(*

## Short summary
This class provides assert statements for bytes.

.. <legal notes>

legal notes
=================
| SPDX-FileCopyrightText: © 2022 ekvip automation GmbH <info@ekvip.de>
| SPDX-License-Identifier: Apache-2.0
| For details check: Apache-2.0_

.. _Apache-2.0: https://www.apache.org/licenses/LICENSE-2.0

.. </legal notes>



*)

{attribute 'reflection'}
FUNCTION_BLOCK INTERNAL ByteAssertions EXTENDS AbstractAssertion IMPLEMENTS IByteAssertions
VAR
END_VAR
VAR CONSTANT
	(* least significant bit *)
	LSB	:BYTE := 16#01;
	(* most significant bit *)
	MSB :BYTE := 16#80;
END_VAR

(*

## Short summary
This assertion method checks if the result current value bitwise ``AND`` mask is equal to the expected value

.. <legal notes>

legal notes
=================
| SPDX-FileCopyrightText: © 2022 ekvip automation GmbH <info@ekvip.de>
| SPDX-License-Identifier: Apache-2.0
| For details check: Apache-2.0_

.. _Apache-2.0: https://www.apache.org/licenses/LICENSE-2.0

.. </legal notes>



*)

METHOD andMaskIsEqualTo
VAR_INPUT
	(* current value to check *)
	currentValue	:BYTE;
	(* 2nd operand for bitwise operation *)
	mask			:BYTE;
	(* expected result after masking *)
	expectedValue	:BYTE;
	(* message if the assertion is false *)
	message			:AssertMessage;
END_VAR
IF ((currentValue AND mask) <> expectedValue) THEN
	THIS^.assertionWasWrong(message, THIS^.getDebugInfo('andMaskIsEqualTo'));
END_IF
END_METHOD

(*

## Short summary
This assertion method checks if the result current value bitwise ``AND`` mask
is not equal to the unexpected value

.. <legal notes>

legal notes
=================
| SPDX-FileCopyrightText: © 2022 ekvip automation GmbH <info@ekvip.de>
| SPDX-License-Identifier: Apache-2.0
| For details check: Apache-2.0_

.. _Apache-2.0: https://www.apache.org/licenses/LICENSE-2.0

.. </legal notes>



*)

METHOD andMaskIsNotEqualTo
VAR_INPUT
	(* current value to check *)
	currentValue	:BYTE;
	(* 2nd operand for bitwise operation *)
	mask			:BYTE;
	(* unexpected result after masking *)
	unexpectedValue	:BYTE;
	(* message if the assertion is false *)
	message			:AssertMessage;
END_VAR
IF ((currentValue AND mask) = unexpectedValue) THEN
	THIS^.assertionWasWrong(message, THIS^.getDebugInfo('andMaskIsNotEqualTo'));
END_IF
END_METHOD

(*

## Short summary
This assertion method checks if the selected bit of current value
is equal to the expected value

.. <legal notes>

legal notes
=================
| SPDX-FileCopyrightText: © 2022 ekvip automation GmbH <info@ekvip.de>
| SPDX-License-Identifier: Apache-2.0
| For details check: Apache-2.0_

.. _Apache-2.0: https://www.apache.org/licenses/LICENSE-2.0

.. </legal notes>



*)

METHOD bitXIsEqualTo
VAR_INPUT
	(* current value to check *)
	currentValue	:BYTE;
	(* number of bit to check *)
	number			:BitNumberByte;
	(* expected value of bit *)
	expectedValue	:BOOL;
	(* message if the assertion is false *)
	message			:AssertMessage;
END_VAR
IF (
	TO_BOOL(
		TO_BYTE(SHL(THIS^.LSB, number))
		AND currentValue
	) <> expectedValue
) THEN
	THIS^.assertionWasWrong(message, THIS^.getDebugInfo('bitXIsEqualTo'));
END_IF
END_METHOD

(*

## Short summary
This assertion method checks if the selected bit of current value
is not equal to the unexpected value

.. <legal notes>

legal notes
=================
| SPDX-FileCopyrightText: © 2022 ekvip automation GmbH <info@ekvip.de>
| SPDX-License-Identifier: Apache-2.0
| For details check: Apache-2.0_

.. _Apache-2.0: https://www.apache.org/licenses/LICENSE-2.0

.. </legal notes>



*)

METHOD bitXIsNotEqualTo
VAR_INPUT
	(* current value to check *)
	currentValue	:BYTE;
	(* number of bit to check *)
	number			:BitNumberByte;
	(* unexpected value of bit *)
	unexpectedValue	:BOOL;
	(* message if the assertion is false *)
	message			:AssertMessage;
END_VAR
IF (
	TO_BOOL(
		TO_BYTE(SHL(THIS^.LSB, number))
		AND currentValue
	) = unexpectedValue
) THEN
	THIS^.assertionWasWrong(message, THIS^.getDebugInfo('bitXIsNotEqualTo'));
END_IF
END_METHOD

(*

## Short summary
This assertion method checks if the selected bit of current value
is set

.. <legal notes>

legal notes
=================
| SPDX-FileCopyrightText: © 2022 ekvip automation GmbH <info@ekvip.de>
| SPDX-License-Identifier: Apache-2.0
| For details check: Apache-2.0_

.. _Apache-2.0: https://www.apache.org/licenses/LICENSE-2.0

.. </legal notes>



*)

METHOD bitXIsSet
VAR_INPUT
	(* current value to check *)
	currentValue	:BYTE;
	(* number of bit to check *)
	number			:BitNumberByte;
	(* message if the assertion is false *)
	message			:AssertMessage;
END_VAR
IF (
	NOT TO_BOOL(
		TO_BYTE(SHL(THIS^.LSB, number))
		AND currentValue
	)
) THEN
	THIS^.assertionWasWrong(message, THIS^.getDebugInfo('bitXIsSet'));
END_IF
END_METHOD

(*

## Short summary
This assertion method checks if the selected bit of current value
is unset

.. <legal notes>

legal notes
=================
| SPDX-FileCopyrightText: © 2022 ekvip automation GmbH <info@ekvip.de>
| SPDX-License-Identifier: Apache-2.0
| For details check: Apache-2.0_

.. _Apache-2.0: https://www.apache.org/licenses/LICENSE-2.0

.. </legal notes>



*)

METHOD bitXIsUnset
VAR_INPUT
	(* current value to check *)
	currentValue	:BYTE;
	(* number of bit to check *)
	number			:BitNumberByte;
	(* message if the assertion is false *)
	message			:AssertMessage;
END_VAR
IF (
	TO_BOOL(
		TO_BYTE(SHL(THIS^.LSB, number))
		AND currentValue
	)
) THEN
	THIS^.assertionWasWrong(message, THIS^.getDebugInfo('bitXIsUnset'));
END_IF
END_METHOD

(*

## Short summary
This abstract property returns the class name of the concrete object, 
It's for debugging purpose

.. <legal notes>

legal notes
=================
| SPDX-FileCopyrightText: © 2022 ekvip automation GmbH <info@ekvip.de>
| SPDX-License-Identifier: Apache-2.0
| For details check: Apache-2.0_

.. _Apache-2.0: https://www.apache.org/licenses/LICENSE-2.0

.. </legal notes>

*)

PROPERTY className :CNM_AbstractObject.ClassName
GET
className := 'CNM_Assertor.ByteAssertions';
END_GET
END_PROPERTY

(*

## Short summary
This assertion method checks if the least significant bit of current value
is equal to the expected value

.. <legal notes>

legal notes
=================
| SPDX-FileCopyrightText: © 2022 ekvip automation GmbH <info@ekvip.de>
| SPDX-License-Identifier: Apache-2.0
| For details check: Apache-2.0_

.. _Apache-2.0: https://www.apache.org/licenses/LICENSE-2.0

.. </legal notes>



*)

METHOD lsbIsEqualTo
VAR_INPUT
	(* current value to check *)
	currentValue	:BYTE;
	(* expected value of lsb *)
	expectedValue	:BOOL;
	(* message if the assertion is false *)
	message			:AssertMessage;
END_VAR
IF (TO_BOOL(currentValue AND THIS^.LSB) <> expectedValue) THEN
	THIS^.assertionWasWrong(message, THIS^.getDebugInfo('lsbIsEqualTo'));
END_IF
END_METHOD

(*

## Short summary
This assertion method checks if the least significant bit of current value
is not equal to the unexpected value

.. <legal notes>

legal notes
=================
| SPDX-FileCopyrightText: © 2022 ekvip automation GmbH <info@ekvip.de>
| SPDX-License-Identifier: Apache-2.0
| For details check: Apache-2.0_

.. _Apache-2.0: https://www.apache.org/licenses/LICENSE-2.0

.. </legal notes>



*)

METHOD lsbIsNotEqualTo
VAR_INPUT
	(* current value to check *)
	currentValue	:BYTE;
	(* unexpected value of lsb *)
	unexpectedValue	:BOOL;
	(* message if the assertion is false *)
	message			:AssertMessage;
END_VAR
IF (TO_BOOL(currentValue AND THIS^.LSB) = unexpectedValue) THEN
	THIS^.assertionWasWrong(message, THIS^.getDebugInfo('lsbIsNotEqualTo'));
END_IF
END_METHOD

(*

## Short summary
This assertion method checks if the least significant bit of current value
is set

.. <legal notes>

legal notes
=================
| SPDX-FileCopyrightText: © 2022 ekvip automation GmbH <info@ekvip.de>
| SPDX-License-Identifier: Apache-2.0
| For details check: Apache-2.0_

.. _Apache-2.0: https://www.apache.org/licenses/LICENSE-2.0

.. </legal notes>



*)

METHOD lsbIsSet
VAR_INPUT
	(* current value to check *)
	currentValue	:BYTE;
	(* message if the assertion is false *)
	message			:AssertMessage;
END_VAR
IF (NOT TO_BOOL(currentValue AND THIS^.LSB)) THEN
	THIS^.assertionWasWrong(message, THIS^.getDebugInfo('lsbIsSet'));
END_IF
END_METHOD

(*

## Short summary
This assertion method checks if the least significant bit of current value
is unset

.. <legal notes>

legal notes
=================
| SPDX-FileCopyrightText: © 2022 ekvip automation GmbH <info@ekvip.de>
| SPDX-License-Identifier: Apache-2.0
| For details check: Apache-2.0_

.. _Apache-2.0: https://www.apache.org/licenses/LICENSE-2.0

.. </legal notes>



*)

METHOD lsbIsUnset
VAR_INPUT
	(* current value to check *)
	currentValue	:BYTE;
	(* message if the assertion is false *)
	message			:AssertMessage;
END_VAR
IF (TO_BOOL(currentValue AND THIS^.LSB)) THEN
	THIS^.assertionWasWrong(message, THIS^.getDebugInfo('lsbIsUnset'));
END_IF
END_METHOD

(*

## Short summary
This assertion method checks if the most significant bit of current value
is equal to the expected value

.. <legal notes>

legal notes
=================
| SPDX-FileCopyrightText: © 2022 ekvip automation GmbH <info@ekvip.de>
| SPDX-License-Identifier: Apache-2.0
| For details check: Apache-2.0_

.. _Apache-2.0: https://www.apache.org/licenses/LICENSE-2.0

.. </legal notes>



*)

METHOD msbIsEqualTo
VAR_INPUT
	(* current value to check *)
	currentValue	:BYTE;
	(* expected value of msb *)
	expectedValue	:BOOL;
	(* message if the assertion is false *)
	message			:AssertMessage;
END_VAR
IF (TO_BOOL(currentValue AND THIS^.MSB) <> expectedValue) THEN
	THIS^.assertionWasWrong(message, THIS^.getDebugInfo('msbIsEqualTo'));
END_IF
END_METHOD

(*

## Short summary
This assertion method checks if the most significant bit of current value
is not equal to the unexpected value

.. <legal notes>

legal notes
=================
| SPDX-FileCopyrightText: © 2022 ekvip automation GmbH <info@ekvip.de>
| SPDX-License-Identifier: Apache-2.0
| For details check: Apache-2.0_

.. _Apache-2.0: https://www.apache.org/licenses/LICENSE-2.0

.. </legal notes>



*)

METHOD msbIsNotEqualTo
VAR_INPUT
	(* current value to check *)
	currentValue	:BYTE;
	(* unexpected value of msb *)
	unexpectedValue	:BOOL;
	(* message if the assertion is false *)
	message			:AssertMessage;
END_VAR
IF (TO_BOOL(currentValue AND THIS^.MSB) = unexpectedValue) THEN
	THIS^.assertionWasWrong(message, THIS^.getDebugInfo('msbIsNotEqualTo'));
END_IF
END_METHOD

(*

## Short summary
This assertion method checks if the most significant bit of current value
is set

.. <legal notes>

legal notes
=================
| SPDX-FileCopyrightText: © 2022 ekvip automation GmbH <info@ekvip.de>
| SPDX-License-Identifier: Apache-2.0
| For details check: Apache-2.0_

.. _Apache-2.0: https://www.apache.org/licenses/LICENSE-2.0

.. </legal notes>



*)

METHOD msbIsSet
VAR_INPUT
	(* current value to check *)
	currentValue	:BYTE;
	(* message if the assertion is false *)
	message			:AssertMessage;
END_VAR
IF (NOT TO_BOOL(currentValue AND THIS^.MSB)) THEN
	THIS^.assertionWasWrong(message, THIS^.getDebugInfo('msbIsSet'));
END_IF
END_METHOD

(*

## Short summary
This assertion method checks if the most significant bit of current value
is unset

.. <legal notes>

legal notes
=================
| SPDX-FileCopyrightText: © 2022 ekvip automation GmbH <info@ekvip.de>
| SPDX-License-Identifier: Apache-2.0
| For details check: Apache-2.0_

.. _Apache-2.0: https://www.apache.org/licenses/LICENSE-2.0

.. </legal notes>



*)

METHOD msbIsUnset
VAR_INPUT
	(* current value to check *)
	currentValue	:BYTE;
	(* message if the assertion is false *)
	message			:AssertMessage;
END_VAR
IF (TO_BOOL(currentValue AND THIS^.MSB)) THEN
	THIS^.assertionWasWrong(message, THIS^.getDebugInfo('msbIsUnset'));
END_IF
END_METHOD

(*

## Short summary
This assertion method checks if the result current value bitwise ``OR`` mask is equal to the expected value

.. <legal notes>

legal notes
=================
| SPDX-FileCopyrightText: © 2022 ekvip automation GmbH <info@ekvip.de>
| SPDX-License-Identifier: Apache-2.0
| For details check: Apache-2.0_

.. _Apache-2.0: https://www.apache.org/licenses/LICENSE-2.0

.. </legal notes>



*)

METHOD orMaskIsEqualTo
VAR_INPUT
	(* current value to check *)
	currentValue	:BYTE;
	(* 2nd operand for bitwise operation *)
	mask			:BYTE;
	(* expected result after masking *)
	expectedValue	:BYTE;
	(* message if the assertion is false *)
	message			:AssertMessage;
END_VAR
IF ((currentValue OR mask) <> expectedValue) THEN
	THIS^.assertionWasWrong(message, THIS^.getDebugInfo('orMaskIsEqualTo'));
END_IF
END_METHOD

(*

## Short summary
This assertion method checks if the result current value bitwise ``OR`` mask 
is not equal to the unexpected value

.. <legal notes>

legal notes
=================
| SPDX-FileCopyrightText: © 2022 ekvip automation GmbH <info@ekvip.de>
| SPDX-License-Identifier: Apache-2.0
| For details check: Apache-2.0_

.. _Apache-2.0: https://www.apache.org/licenses/LICENSE-2.0

.. </legal notes>



*)

METHOD orMaskIsNotEqualTo
VAR_INPUT
	(* current value to check *)
	currentValue	:BYTE;
	(* 2nd operand for bitwise operation *)
	mask			:BYTE;
	(* unexpected result after masking *)
	unexpectedValue	:BYTE;
	(* message if the assertion is false *)
	message			:AssertMessage;
END_VAR
IF ((currentValue OR mask) = unexpectedValue) THEN
	THIS^.assertionWasWrong(message, THIS^.getDebugInfo('orMaskIsNotEqualTo'));
END_IF
END_METHOD

(*

## Short summary
This assertion method checks if the current value is equal to the expected value

.. <legal notes>

legal notes
=================
| SPDX-FileCopyrightText: © 2022 ekvip automation GmbH <info@ekvip.de>
| SPDX-License-Identifier: Apache-2.0
| For details check: Apache-2.0_

.. _Apache-2.0: https://www.apache.org/licenses/LICENSE-2.0

.. </legal notes>



*)

METHOD valueIsEqualTo
VAR_INPUT
	(* current value to check *)
	currentValue	:BYTE;
	(* expected value to compare *)
	expectedValue	:BYTE;
	(* message if the assertion is false *)
	message			:AssertMessage;
END_VAR
IF (currentValue <> expectedValue) THEN
	THIS^.assertionWasWrong(message, THIS^.getDebugInfo('valueIsEqualTo'));
END_IF
END_METHOD

(*

## Short summary
This assertion method checks if the current value is greater than the less value

.. <legal notes>

legal notes
=================
| SPDX-FileCopyrightText: © 2022 ekvip automation GmbH <info@ekvip.de>
| SPDX-License-Identifier: Apache-2.0
| For details check: Apache-2.0_

.. _Apache-2.0: https://www.apache.org/licenses/LICENSE-2.0

.. </legal notes>



*)

METHOD valueIsGreaterThan
VAR_INPUT
	(* current value to check *)
	currentValue	:BYTE;
	(* less than lower limit *)
	lessValue		:BYTE;
	(* message if the assertion is false *)
	message			:AssertMessage;
END_VAR
IF (currentValue <= lessValue) THEN
	THIS^.assertionWasWrong(message, THIS^.getDebugInfo('valueIsGreaterThan'));
END_IF
END_METHOD

(*

## Short summary
This assertion method checks if the current value is inside a limit

**Attention:** 
	limits are included: ``valueIsInRangeOf(3, 3, 3)`` is a true assertion

.. <legal notes>

legal notes
=================
| SPDX-FileCopyrightText: © 2022 ekvip automation GmbH <info@ekvip.de>
| SPDX-License-Identifier: Apache-2.0
| For details check: Apache-2.0_

.. _Apache-2.0: https://www.apache.org/licenses/LICENSE-2.0

.. </legal notes>



*)

METHOD valueIsInRangeOf
VAR_INPUT
	(* lower limit for the current value *)
	lowerLimit		:BYTE;
	(* current value to check *)
	currentValue	:BYTE;
	(* upper limit for the current value *)
	upperLimit		:BYTE;
	(* message if the assertion is false *)
	message			:AssertMessage;
END_VAR
IF (
	(currentValue < lowerLimit)
	OR (currentValue > upperLimit)
) THEN
	THIS^.assertionWasWrong(message, THIS^.getDebugInfo('valueIsInRangeOf'));
END_IF
END_METHOD

(*

## Short summary
This assertion method checks if the current value is less than the greater value

.. <legal notes>

legal notes
=================
| SPDX-FileCopyrightText: © 2022 ekvip automation GmbH <info@ekvip.de>
| SPDX-License-Identifier: Apache-2.0
| For details check: Apache-2.0_

.. _Apache-2.0: https://www.apache.org/licenses/LICENSE-2.0

.. </legal notes>



*)

METHOD valueIsLessThan
VAR_INPUT
	(* current value to check *)
	currentValue	:BYTE;
	(* greater than upper limit *)
	greaterValue	:BYTE;
	(* message if the assertion is false *)
	message			:AssertMessage;
END_VAR
IF (currentValue >= greaterValue) THEN
	THIS^.assertionWasWrong(message, THIS^.getDebugInfo('valueIsLessThan'));
END_IF
END_METHOD

(*

## Short summary
This assertion method checks if the current value is less than or equal to the maximum value

.. <legal notes>

legal notes
=================
| SPDX-FileCopyrightText: © 2022 ekvip automation GmbH <info@ekvip.de>
| SPDX-License-Identifier: Apache-2.0
| For details check: Apache-2.0_

.. _Apache-2.0: https://www.apache.org/licenses/LICENSE-2.0

.. </legal notes>



*)

METHOD valueIsMax
VAR_INPUT
	(* current value to check *)
	currentValue	:BYTE;
	(* upper limit for the current value *)
	maximumValue	:BYTE;
	(* message if the assertion is false *)
	message			:AssertMessage;
END_VAR
IF (currentValue > maximumValue) THEN
	THIS^.assertionWasWrong(message, THIS^.getDebugInfo('valueIsMax'));
END_IF
END_METHOD

(*

## Short summary
This assertion method checks if the current value is greater than or equal to the minimum value

.. <legal notes>

legal notes
=================
| SPDX-FileCopyrightText: © 2022 ekvip automation GmbH <info@ekvip.de>
| SPDX-License-Identifier: Apache-2.0
| For details check: Apache-2.0_

.. _Apache-2.0: https://www.apache.org/licenses/LICENSE-2.0

.. </legal notes>



*)

METHOD valueIsMin
VAR_INPUT
	(* current value to check *)
	currentValue	:BYTE;
	(* lower limit for the current value *)
	minimumValue	:BYTE;
	(* message if the assertion is false *)
	message			:AssertMessage;
END_VAR
IF (currentValue < minimumValue) THEN
	THIS^.assertionWasWrong(message, THIS^.getDebugInfo('valueIsMin'));
END_IF
END_METHOD

(*

## Short summary
This assertion method checks if the current value is not equal to the unexpected value

.. <legal notes>

legal notes
=================
| SPDX-FileCopyrightText: © 2022 ekvip automation GmbH <info@ekvip.de>
| SPDX-License-Identifier: Apache-2.0
| For details check: Apache-2.0_

.. _Apache-2.0: https://www.apache.org/licenses/LICENSE-2.0

.. </legal notes>



*)

METHOD valueIsNotEqualTo
VAR_INPUT
	(* current value to check *)
	currentValue	:BYTE;
	(* unexpected value to compare *)
	unexpectedValue	:BYTE;
	(* message if the assertion is false *)
	message			:AssertMessage;
END_VAR
IF (currentValue = unexpectedValue) THEN
	THIS^.assertionWasWrong(message, THIS^.getDebugInfo('valueIsNotEqualTo'));
END_IF
END_METHOD

(*

## Short summary
This assertion method checks if the result current value bitwise ``XOR`` mask is equal to the expected value

.. <legal notes>

legal notes
=================
| SPDX-FileCopyrightText: © 2022 ekvip automation GmbH <info@ekvip.de>
| SPDX-License-Identifier: Apache-2.0
| For details check: Apache-2.0_

.. _Apache-2.0: https://www.apache.org/licenses/LICENSE-2.0

.. </legal notes>



*)

METHOD xorMaskIsEqualTo
VAR_INPUT
	(* current value to check *)
	currentValue	:BYTE;
	(* 2nd operand for bitwise operation *)
	mask			:BYTE;
	(* expected result after masking *)
	expectedValue	:BYTE;
	(* message if the assertion is false *)
	message			:AssertMessage;
END_VAR
IF ((currentValue XOR mask) <> expectedValue) THEN
	THIS^.assertionWasWrong(message, THIS^.getDebugInfo('xorMaskIsEqualTo'));
END_IF
END_METHOD

(*

## Short summary
This assertion method checks if the result current value bitwise ``XOR`` mask 
is not equal to the unexpected value

.. <legal notes>

legal notes
=================
| SPDX-FileCopyrightText: © 2022 ekvip automation GmbH <info@ekvip.de>
| SPDX-License-Identifier: Apache-2.0
| For details check: Apache-2.0_

.. _Apache-2.0: https://www.apache.org/licenses/LICENSE-2.0

.. </legal notes>



*)

METHOD xorMaskIsNotEqualTo
VAR_INPUT
	(* current value to check *)
	currentValue	:BYTE;
	(* 2nd operand for bitwise operation *)
	mask			:BYTE;
	(* unexpected result after masking *)
	unexpectedValue	:BYTE;
	(* message if the assertion is false *)
	message			:AssertMessage;
END_VAR
IF ((currentValue XOR mask) = unexpectedValue) THEN
	THIS^.assertionWasWrong(message, THIS^.getDebugInfo('xorMaskIsNotEqualTo'));
END_IF
END_METHOD

END_FUNCTION_BLOCK

(* stored: Version 1.1.0.1, ProductVersion 3.1.4026.11
   POU ByteAssertions: Id {3e37a8d1-5228-401d-b4c2-725f42cb4975}, SpecialFunc None
   Method andMaskIsEqualTo: Id {c6103606-cb33-4a26-aca7-82030cf004ff}
   Method andMaskIsNotEqualTo: Id {b348b00b-4543-446e-a9e3-dc5347f8443c}
   Method bitXIsEqualTo: Id {815ab244-174f-4642-afda-0202ba21352f}
   Method bitXIsNotEqualTo: Id {0cd4a95d-9189-48ae-885c-2777876e3b37}
   Method bitXIsSet: Id {32ea1839-133f-41e8-840b-46460d45ffe9}
   Method bitXIsUnset: Id {0d16ef69-6b4a-4914-a653-3e8b87a6afe6}
   Property className: Id {14e55640-849a-42ad-bc9b-b5f023055877}
   Get Get: Id {8a414597-5774-49ed-9d75-5245bdb706d7}
   Method lsbIsEqualTo: Id {a64aa9c5-02df-4703-85fb-780af0d86264}
   Method lsbIsNotEqualTo: Id {260f6cc6-b807-46db-8f04-22aa5481e4dc}
   Method lsbIsSet: Id {a46dc1b5-b5d2-4d0e-9000-919c626056a6}
   Method lsbIsUnset: Id {cb63d466-4fa9-497b-a442-1b1f13a847ad}
   Method msbIsEqualTo: Id {0d24647c-3f05-408a-8ce2-1f14d228f9bf}
   Method msbIsNotEqualTo: Id {9b2e751a-1a56-43b1-a1bc-fb3bafe2e8f8}
   Method msbIsSet: Id {6ebf6619-d290-4308-9e8a-68550de60f9f}
   Method msbIsUnset: Id {e99ddac1-b61e-407f-8dec-70150db5c955}
   Method orMaskIsEqualTo: Id {87959efa-58ab-4fc4-a587-78228fa25d7f}
   Method orMaskIsNotEqualTo: Id {474506ea-ae02-43e7-840f-a343500164ea}
   Method valueIsEqualTo: Id {f35bbdfe-87cb-4b61-9879-884720709b7e}
   Method valueIsGreaterThan: Id {33e281ff-e801-407b-b8dd-cb8127560a58}
   Method valueIsInRangeOf: Id {69e93f1b-91ea-45a4-9ca8-fab4921639d0}
   Method valueIsLessThan: Id {7f70c044-0ae6-4285-9705-07fdba8b0777}
   Method valueIsMax: Id {51d5ab79-7b26-4136-b1b9-d686ac6a7e4d}
   Method valueIsMin: Id {f3bfb5e9-f6f3-450b-862b-d2dcb7eca397}
   Method valueIsNotEqualTo: Id {11264ce5-ab55-4399-8313-63a75ca37b35}
   Method xorMaskIsEqualTo: Id {3e9b699b-6253-4376-94f9-90a90fda06d4}
   Method xorMaskIsNotEqualTo: Id {691fa9b3-96df-4c42-99d7-88d2411fa92f} *)
